// TwinCAT 3 PLC project Printing_Controller
// ProgramVersion: 3.1.4024.0
// libraries:
//   Tc2_Standard, * (Beckhoff Automation GmbH)
//   Tc2_System, * (Beckhoff Automation GmbH)
//   Tc3_Module, * (Beckhoff Automation GmbH)
// project tree:
//   GVLs/ GVL.TcGVL, GVL_IO.TcGVL, GVL_LAP.TcGVL, README.TcGVL
//   / PlcTask.TcTTO
//   POUs/Component/ P_CC1_Enable.TcPOU, P_CP1_Check.TcPOU, P_CP1_Enable.TcPOU
//   POUs/ FB_SetConfigData.TcPOU, FB_GetOutputData.TcPOU, FB_SetOutPutDataToIO.TcPOU, MAIN.TcPOU, P_Control_Mode.TcPOU, P_Laptop_Operate.TcPOU, P_Robot_Operate.TcPOU
//   POUs/Utils/ F_LowpassFilter.TcPOU, F_ScalAnalogOut.TcPOU
// real-time tasks:
//   TASK PlcTask: cycle T#10ms, priority 20, ADS port 350
// I/O:
//   DEVICE Device 1 (EtherCAT), AmsNetId 5.151.68.134.2.1
//     Term 1 (EK1200) [EK1200-5000 EtherCAT Power supply (2A E-Bus)]
//       Term 2 (EL1008) [EL1008 8Ch. Dig. Input 24V, 3ms]
//       Term 3 (EL2008) [EL2008 8Ch. Dig. Output 24V, 0.5A]
//       Term 4 (EL3014) [EL3014 4Ch. Ana. Input 0-20mA DIFF]
//       Term 5 (EL4134) [EL4134 4Ch. Ana. Output -10/+10V, 16bit]
//       Term 6 (EL6631-0010) [EL6631-0010 PROFINET IO Device]
//       Term 7 (EL9011) [EL9011 End Terminal]
// variable links:
//   Printing_Controller/Printing_Controller Instance <-> Device 1 (EtherCAT)/Term 1 (EK1200)/Term 2 (EL1008)
//     PlcTask Inputs/GVL_IO.ibSpare1 <-> Channel 5/Input
//     PlcTask Inputs/GVL_IO.ib_CC1_Button_Mode_Laptop <-> Channel 8/Input
//     PlcTask Inputs/GVL_IO.ib_CC1_Button_Mode_Manual <-> Channel 6/Input
//     PlcTask Inputs/GVL_IO.ib_CC1_Button_Reset <-> Channel 7/Input
//     PlcTask Inputs/GVL_IO.ib_CC1_Safety_Ready <-> Channel 1/Input
//     PlcTask Inputs/GVL_IO.ib_CP1_Drive_Error <-> Channel 4/Input
//     PlcTask Inputs/GVL_IO.ib_CP1_Ready <-> Channel 3/Input
//     PlcTask Inputs/GVL_IO.ib_CP1_Safety_Grid_Mounted <-> Channel 2/Input
//   Printing_Controller/Printing_Controller Instance <-> Device 1 (EtherCAT)/Term 1 (EK1200)/Term 3 (EL2008)
//     PlcTask Outputs/GVL_IO.ob_CC1_Safety_Reset <-> Channel 1/Output
//     PlcTask Outputs/GVL_IO.ob_CP1_Backward <-> Channel 5/Output
//     PlcTask Outputs/GVL_IO.ob_CP1_Forward <-> Channel 4/Output
//     PlcTask Outputs/GVL_IO.ob_CP1_Start <-> Channel 3/Output
//     PlcTask Outputs/GVL_IO.ob_CP1_Stop <-> Channel 2/Output
//   Printing_Controller/Printing_Controller Instance <-> Device 1 (EtherCAT)/Term 1 (EK1200)/Term 4 (EL3014)
//     PlcTask Inputs/GVL_IO.ib_CP1_Actual_Speed <-> AI Standard Channel 1/Value
//   Printing_Controller/Printing_Controller Instance <-> Device 1 (EtherCAT)/Term 1 (EK1200)/Term 5 (EL4134)
//     PlcTask Outputs/GVL_IO.on_CP1_Speed <-> AO Output Channel 1/Analog output

CONFIGURATION Printing_Controller
    RESOURCE PLC ON TwinCAT3
        TASK PlcTask(INTERVAL := T#10ms, PRIORITY := 20);
        PROGRAM MAIN WITH PlcTask : MAIN;
    END_RESOURCE
END_CONFIGURATION

// ---- GVLs/GVL.TcGVL
{attribute 'qualified_only'}
// ***********************************************************************************
//
// USI Mendrisio, Largo Bernasconi 2, CH-6850 Mendrisio
// ETH Zurich, Building HIF E26, Laura-Hezner-Weg 7, CH-8093 Zürich
// 
// ***********************************************************************************
// 
// PROJECT     :  Clay Printing Controller
// FUNCTION    :  Global varable
// AUTHOR      :  WeiTing Chen
// EMAIL       :  chen@mesh.ch
// Copyright   :  USI FMAA Mendrisio(CH) 2025
//
// ***********************************************************************************


VAR_GLOBAL
	
	// Controller 1
	b_mode_manual : BOOL;
	b_mode_laptop : BOOL; 
	b_mode_robot : BOOL;  
	
	b_CC1_enable :BOOL;
	b_CC1_power_on: BOOL;
	s_current_mode: STRING;
	
	// Machine 1
	// Machine 2
	
	// Concrete Pump 1
	b_CP1_Check_On : BOOL;
	b_CP1_is_run : BOOL;
	b_CP1_is_ready : BOOL;	
	b_CP1_power_on :BOOL;
	b_CP1_safety_grid_on : BOOL;
	b_CP1_drive_error :BOOL;
	
	
	// Config
	// Concrete Pump 1
	f_CP1_Max_Flowrate : REAL;
	f_CP1_Check_Flowrate : REAL;
	t_CP1_Check_Duration : TIME;
 	n_CP1_Flush_Flowrate :REAL;	
	
END_VAR

// ---- GVLs/GVL_IO.TcGVL
{attribute 'qualified_only'}

// ***********************************************************************************
//
// USI Mendrisio, Largo Bernasconi 2, CH-6850 Mendrisio
// ETH Zurich, Building HIF E26, Laura-Hezner-Weg 7, CH-8093 Zürich
//
// ***********************************************************************************
//
// PROJECT     :  Clay Printing Controller
// FUNCTION    :  Global Hareware IO
// AUTHOR      :  WeiTing Chen
// EMAIL       :  chen@mesh.ch
// Copyright   :  USI FMAA Mendrisio(CH) 2025
//
// ***********************************************************************************

VAR_GLOBAL

	// ***** HARDWARE INPUT ******

	// Concrete Controller 1
	// This once install the safety gate, we can start to do read from it.
	ib_CC1_Safety_Ready_NOT_IMP AT %I*: BOOL;  // DI1
	ib_CC1_Safety_Ready:BOOL;
	ib_CC1_Button_Mode_Manual   AT %I*: BOOL;  // DI6
	ib_CC1_Button_Mode_Laptop   AT %I*: BOOL;  // DI8
	ib_CC1_Button_Reset         AT %I*: BOOL;  // DI7

	// Concrete Pump 1
	ib_CP1_Safety_Grid_Mounted  AT %I*: BOOL;  // DI2
	ib_CP1_Ready                AT %I*: BOOL;  // DI3
	ib_CP1_Drive_Error          AT %I*: BOOL;  // DI4
	ib_CP1_Actual_Speed         AT %I*: INT;   // AI1

	// Spare Slot
	ibSpare1 AT %I*: BOOL;  //DI5
	inSpare2 AT %I*: INT;   //AI2
	inSpare3 AT %I*: INT;   //AI3
	inSpare4 AT %I*: INT;   //AI4


	// ***** HARDWARE OUTPUT ******

	// Concrete Controller 1
	ob_CC1_Safety_Reset AT %Q*: BOOL;  //DO1

	// Concrete Pump 1
	ob_CP1_Start    AT %Q*: BOOL;  //DO3
	ob_CP1_Stop     AT %Q*: BOOL;  //DO2
	ob_CP1_Forward  AT %Q*: BOOL;  //DO4
	ob_CP1_Backward AT %Q*: BOOL;  //DO5
	on_CP1_Speed    AT %Q*: INT;   //AO1
	// just for testing, if not working after we can delete it.
	on_CP1_Speed_test    AT %Q*: INT;   //AOTemp

	// Spare Slot
	obSpare6 AT %Q*: BOOL;  //DO6
	obSpare7 AT %Q*: BOOL;  //DO7
	obSpare8 AT %Q*: BOOL;  //DO8

	onSpare2 AT %Q*: INT;   //AO2
	onSpare3 AT %Q*: INT;   //AO3
	onSpare4 AT %Q*: INT;   //AO4

END_VAR

// ---- GVLs/GVL_LAP.TcGVL
{attribute 'qualified_only'}

// ***********************************************************************************
//
// USI Mendrisio, Largo Bernasconi 2, CH-6850 Mendrisio
// ETH Zurich, Building HIF E26, Laura-Hezner-Weg 7, CH-8093 Zürich
//
// ***********************************************************************************
//
// PROJECT     :  Clay Printing Controller
// FUNCTION    :  Global Laptop IO wrapper
// AUTHOR      :  WeiTing Chen
// EMAIL       :  chen@mesh.ch
// Copyright   :  USI FMAA Mendrisio(CH) 2025
//
// ***********************************************************************************

VAR_GLOBAL
	
	CONCRETE_CONTROLLER: STRING := 'Controller'; //*****
	b_Operate_mode_manual             : BOOL;
	b_Operate_mode_laptop             : BOOL;
	b_Operate_mode_robot              : BOOL;
	b_Concrete_Controller_enable      : BOOL;
	b_Concrete_Controller_reset       : BOOL;
	b_Concrete_Controller_power_on    : BOOL;
	n_Concrete_Controller_current_mode: INT;
	
	CONCRETE_PUMP: STRING := 'CONCRETE_PUMP'; //*****
	// Concrete Pump
	// input
	
	b_Concrete_Pump_Power_On   : BOOL;  // Power On
	b_Concrete_Pump_Forward_On : BOOL;  // Forward ON
	b_Concrete_Pump_Backward_On: BOOL;  // Backward ON
	
	b_Concrete_Pump_Flush_On      : BOOL;  // FLUSH MODE ON
	n_Concrete_Pump_Flush_Flowrate: REAL;  // READ [l/min]
	
	b_Concrete_Pump_Check_On      : BOOL;       // CHECK MODE ON
	
	// TODO: Need to check the range of flowrate
	f_Concrete_Pump_Check_Flowrate: REAL;       // [O tp 24 l/min]
	n_Concrete_Pump_Check_Duration: INT := 15;  // [s]
	
	f_Concrete_Pump_Set_Flowrate : REAL;          // [0 to 24 l/min]
	f_Concrete_Pump_dosing_volume: REAL := 0.32;  // calibrated XXXXX
	n_Concrete_Pump_Max_Speed    : INT := 75;     // calibrated XXXXX
	n_Concrete_Pump_Set_Speed    : INT;           // WRITE VALUE From 0 to 75 [rpm]
	
	
	b_CP1_is_run        : BOOL;
	b_CP1_is_ready      : BOOL;
	b_CP1_power_on      : BOOL;
	b_CP1_safety_grid_on: BOOL;
	b_CP1_drive_error   : BOOL;
	
	
	f_CP1_status_torque :REAL;
	f_CP1_status_speed: REAL;
	
	// Other
	Admixture_Pump_1: STRING := 'Admixture Pump (AP1)'; //*****

END_VAR

// ---- GVLs/README.TcGVL
{attribute 'qualified_only'}
// ***********************************************************************************
//
// USI Mendrisio, Largo Bernasconi 2, CH-6850 Mendrisio
// ETH Zurich, Building HIF E26, Laura-Hezner-Weg 7, CH-8093 Zürich
//
// ***********************************************************************************
//
// PROJECT     :  Clay Printing Controller
// FUNCTION    :  README
// AUTHOR      :  WeiTing Chen
// EMAIL       :  chen@mesh.ch
// Copyright   :  USI FMAA Mendrisio(CH) 2025
//
// ***********************************************************************************

VAR_GLOBAL
(*
Set the IP with XXXXXXXX

File description
GVL(GVL : Global variables)
GVL_IO(GVL_IO : IO)
GVL_LAP(GVL_LAP : variables for control via laptop)

Data Type Prefix
ib = Input Bool   / ob = Output Bool
if = Input float  / of = Output float (REAL, LREAL)
in = Input numeric/ on = Output numeric
(INT, SINT, USINT, UNIT, DINT, UDINT, BYTE, WORD, DWORD, LWORD, XINT, UXINT, XWORD)
t = Time (TON)
s = String

Naming Shortcuts
CC1 = Concrete Controller
CP1 = Concrete Pump
PN = Profinet with Roboter

*)
END_VAR

// ---- POUs/MAIN.TcPOU
PROGRAM MAIN
VAR
END_VAR


// ***********************************************************************************
//
// USI Mendrisio, Largo Bernasconi 2, CH-6850 Mendrisio
// ETH Zurich, Building HIF E26, Laura-Hezner-Weg 7, CH-8093 Zürich
//
// ***********************************************************************************
//
// PROJECT     :  Clay Printing Controller
// FUNCTION    :  Main
// AUTHOR      :  WeiTing Chen
// EMAIL       :  chen@mesh.ch
// Copyright   :  USI FMAA Mendrisio(CH) 2025
//
// ***********************************************************************************


// Control Mode select
P_Control_Mode();

// Operation Mode select
// TODO: Implementation of the operation mode. Now everything services as laptop mode.
IF GVL.b_mode_laptop THEN
	P_Laptop_Operate();
ELSIF GVL.b_mode_robot THEN
	P_Laptop_Operate();
ELSIF GVL.b_mode_manual THEN
	P_Laptop_Operate();
END_IF

END_PROGRAM

// ---- POUs/P_Control_Mode.TcPOU
PROGRAM P_Control_Mode
VAR
END_VAR


// ***********************************************************************************
//
// USI Mendrisio, Largo Bernasconi 2, CH-6850 Mendrisio
// ETH Zurich, Building HIF E26, Laura-Hezner-Weg 7, CH-8093 Zürich
//
// ***********************************************************************************
//
// PROJECT     :  Clay Printing Controller
// FUNCTION    :  Control mode selection
// AUTHOR      :  WeiTing Chen
// EMAIL       :  chen@mesh.ch
// Copyright   :  USI FMAA Mendrisio(CH) 2025
//
// ***********************************************************************************


GVL.b_mode_manual := GVL_IO.ib_CC1_Button_Mode_Manual;
GVL.b_mode_laptop := GVL_IO.ib_CC1_Button_Mode_Laptop;
GVL.b_mode_robot := False;

IF GVL.b_mode_manual THEN
	GVL.s_current_mode := 'Controller';
ELSIF GVL.b_mode_laptop  THEN
	GVL.s_current_mode := 'Laptop';
ELSIF NOT GVL.b_mode_manual AND NOT GVL.b_mode_laptop THEN
	GVL.s_current_mode := 'Robot';
	GVL.b_mode_robot := TRUE;
ELSE
	GVL.s_current_mode := 'None';

END_IF

END_PROGRAM

// ---- POUs/P_Laptop_Operate.TcPOU
PROGRAM P_Laptop_Operate
VAR
	SafetyReset 	: bool;
	b_Enable		: BOOL;
	b_Reset			: BOOL;

	fb_SetOutputDataToIO : FB_SetOutputDataToIO;
	fb_getOutputData : FB_GetOutputData;
	fb_setConfig : FB_SetConfigData;

	b_Safety_Reset : BOOL;
	b_Timer_Rest : BOOL;
	t_CC1_Time_Safety_Rest : TIME :=T#5S; //wait 5s for controller restart
	fb_CC1_Trigger_Safety_On : R_TRIG;
	fb_CC1_Trigger_Safety_Off : R_TRIG;
	fb_CC1_Timer_Safety: TON;

END_VAR


// ***********************************************************************************
//
// USI Mendrisio, Largo Bernasconi 2, CH-6850 Mendrisio
// ETH Zurich, Building HIF E26, Laura-Hezner-Weg 7, CH-8093 Zürich
//
// ***********************************************************************************
//
// PROJECT     :  Clay Printing Controller
// FUNCTION    :  Control mode selection
// AUTHOR      :  WeiTing Chen
// EMAIL       :  chen@mesh.ch
// Copyright   :  USI FMAA Mendrisio(CH) 2025
//
// ***********************************************************************************

// Controller reset trigger
b_Timer_Rest:=GVL_LAP.b_Concrete_Controller_reset;

fb_CC1_Timer_Safety(
					IN:=b_Timer_Rest,
					PT:=t_CC1_Time_Safety_Rest);

fb_CC1_Trigger_Safety_On(clk:=fb_CC1_Timer_Safety.IN);
fb_CC1_Trigger_Safety_Off(clk:=fb_CC1_Timer_Safety.Q);
//b_Safety_Reset:=FALSE;
IF fb_CC1_Trigger_Safety_On.Q THEN
	b_Safety_Reset:=TRUE;
END_IF
IF fb_CC1_Trigger_Safety_Off.Q THEN
	b_Safety_Reset:=FALSE;
	GVL_LAP.b_Concrete_Controller_reset:=FALSE;
END_IF
GVL_IO.ob_CC1_Safety_Reset:= b_Safety_Reset OR GVL_IO.ib_CC1_Button_Reset;

// Concrete Controller enable
P_CC1_Enable( b_set_run:= GVL_LAP.b_Concrete_Controller_enable );


//***********************************************************************************
// Set Process Configuration
//***********************************************************************************

fb_setConfig(
// Geneal
// Concrete Controller

// Concrete Pump
_f_CP1_Max_Flowrate   := INT_TO_REAL(GVL_LAP.n_Concrete_Pump_Max_Speed) * GVL_LAP.f_Concrete_Pump_dosing_volume,
_f_CP1_Check_Flowrate := GVL_LAP.f_Concrete_Pump_Check_Flowrate,
_t_CP1_Check_Duration := INT_TO_TIME(GVL_LAP.n_Concrete_Pump_Check_Duration)*1000,

);

//***********************************************************************************
// Setup IO data to PLC
//***********************************************************************************
fb_SetOutputDataToIO(

	// Concrete Pump
	b_CP1_Forward_On       := GVL_LAP.b_Concrete_Pump_Forward_On,
	b_CP1_Backward_On      := GVL_LAP.b_Concrete_Pump_Backward_On,
	b_CP1_Flush_On         := GVL_LAP.b_Concrete_Pump_Flush_On,
	b_CP1_Check_On         := GVL_LAP.b_Concrete_Pump_Check_On,
	n_CP_Flowrate_mode     := TRUE,
	n_CP1_Operate_Flowrate := REAL_TO_UDINT(GVL_LAP.f_Concrete_Pump_Set_Flowrate*100),
	n_CP1_Check_Flowrate   := REAL_TO_UDINT(GVL_LAP.f_Concrete_Pump_Check_Flowrate*100),
	n_CP1_Flush_Flowrate   := REAL_TO_UDINT(GVL_LAP.n_Concrete_Pump_Flush_Flowrate*100),
	f_dosing_volume        := REAL_TO_INT(GVL_LAP.f_concrete_pump_dosing_volume*100),
	n_cp1_max_speed        := GVL_LAP.n_concrete_pump_max_speed,
	n_cp1_target_speed     := GVL_LAP.n_concrete_pump_set_speed,

  //
	);


//***********************************************************************************
// Concrete Pump
//***********************************************************************************

// concrete pump power control is from pump itself
P_CP1_Enable();
P_CP1_Check(b_set_run := fb_SetOutputDataToIO.b_CP1_Forward_On,
			b_check_mode_on  := fb_SetOutputDataToIO.b_CP1_Check_On,
			t_check_duration := fb_setConfig._t_CP1_Check_Duration,
			);


//***********************************************************************************
// Other Pump
//***********************************************************************************

// Put Other pump control here


//***********************************************************************************
// Get out put data from PLC
//***********************************************************************************
fb_getOutputData(

	//CC1
	b_mode_manual := GVL_LAP.b_Operate_mode_manual,
	b_mode_laptop := GVL_LAP.b_Operate_mode_laptop,
	b_mode_robot   := GVL_LAP.b_Operate_mode_robot,
	b_CC1_power_on := GVL_LAP.b_Concrete_Controller_power_on,
	n_current_mode := GVL_LAP.n_Concrete_Controller_current_mode,

	//CP1
	b_CP1_is_run   := GVL_LAP.b_CP1_is_run,
	b_CP1_is_ready := GVL_LAP.b_CP1_is_ready,

	b_CP1_power_on       := GVL_LAP.b_CP1_power_on,
	b_CP1_safety_grid_on := GVL_LAP.b_CP1_safety_grid_on,
	b_CP1_drive_error    := GVL_LAP.b_CP1_drive_error,
	
	f_CP1_status_torque := GVL_LAP.f_CP1_status_torque,
	f_CP1_status_speed := GVL_LAP.f_CP1_status_speed,

);

END_PROGRAM

// ---- POUs/FB_SetOutPutDataToIO.TcPOU
FUNCTION_BLOCK  FB_SetOutPutDataToIO
VAR_INPUT

	// Concrete Pump
	b_CP1_Forward_On : BOOL;
	b_CP1_Backward_On : BOOL;
	b_CP1_Flush_On :BOOL;
	b_CP1_Check_On : BOOL;
	n_CP_Flowrate_mode : BOOL;
	n_CP1_Operate_Flowrate : UDINT;
	n_CP1_Check_Flowrate : UDINT;
	n_CP1_Flush_Flowrate : UDINT;
	f_dosing_volume:INT;

	n_CP1_max_speed : INT ;  // rpm
	n_CP1_target_speed: INT; // rpm

	// Example for AP1
	(*
	b_AP1_Power_On : BOOL;
	b_AP1_Run : BOOL;
	b_AP1_Flush_On :BOOL;
	b_AP1_Check_On :BOOL;

	n_AP1_Flowrate_mode : BOOL;
	n_AP1_Max_Flowrate : INT;
	n_AP1_Operate_Flowrate : UDINT;
	n_AP1_Check_Flowrate : UDINT;
	n_AP1_Flush_Flowrate : UDINT;
	n_AP1_Dosing_factor : INT;
	*)


END_VAR
VAR_OUTPUT
END_VAR
VAR
	// Condition
	_n_temp_flowrate_CP1 : UDINT;
	_n_temp_speed_CP1: INT;

END_VAR

// ***********************************************************************************
//
// USI Mendrisio, Largo Bernasconi 2, CH-6850 Mendrisio
// ETH Zurich, Building HIF E26, Laura-Hezner-Weg 7, CH-8093 Zürich
//
// ***********************************************************************************
//
// PROJECT     :  Clay Printing Controller
// FUNCTION    :  Set data to IO and process (Custom function block)
// AUTHOR      :  WeiTing Chen
// EMAIL       :  chen@mesh.ch
// Copyright   :  USI FMAA Mendrisio(CH) 2025
//
// ***********************************************************************************


// ***********************************************************************************
// Concrete Pump 1
// ***********************************************************************************


// Start
IF  P_CP1_Enable.n_Step=20 THEN
	GVL_IO.ob_CP1_Start:=TRUE;
ELSE
	GVL_IO.ob_CP1_Start:=FALSE;
END_IF

// Stop
IF  P_CP1_Enable.n_Step=40 THEN
	GVL_IO.ob_CP1_Stop:=TRUE;
ELSE
	GVL_IO.ob_CP1_Stop:=FALSE;
END_IF

GVL_IO.ob_CP1_Forward := b_CP1_Forward_On; // Forward
GVL_IO.ob_CP1_Backward := b_CP1_Backward_On; // Backward

// Set speed for pump
IF b_CP1_Flush_On THEN
	//
	// Process speed for flushing or filling the pipe
	 _n_temp_flowrate_CP1:=n_CP1_Flush_Flowrate;
ELSIF P_CP1_Check.n_Step=20 OR P_CP1_Check.n_Step=25 THEN
	//
	// Check Flowrate for pump
	_n_temp_flowrate_CP1 :=n_CP1_Check_Flowrate;
ELSE
	//
	// Process speed for pump
	_n_temp_flowrate_CP1 :=n_CP1_Operate_Flowrate;
END_IF


// Concrete pump speed  0 (0V) to 75 rpm (10V)
IF NOT n_CP_Flowrate_mode THEN
	// set from rpm
	GVL_IO.on_CP1_Speed:=F_ScalAnalogOut(
		n_Input:= INT_TO_UDINT(n_CP1_target_speed),
		n_InMin:= 0,
		n_InMax:= INT_TO_UDINT(n_CP1_max_speed),
		n_OutMin:= 0,
		n_OutMax:= 32767);
ELSE
	// set from flowrate
	GVL_IO.on_CP1_Speed:=F_ScalAnalogOut(
		n_Input:= _n_temp_flowrate_CP1,
		n_InMin:= 0,
		n_InMax:= INT_TO_UDINT(n_CP1_max_speed*f_dosing_volume),
		n_OutMin:= 0,
		n_OutMax:= 32767);
END_IF


//***********************************************************************************
// Other Pump
//***********************************************************************************

END_FUNCTION_BLOCK

// ---- POUs/Component/P_CP1_Enable.TcPOU
PROGRAM P_CP1_Enable
VAR_INPUT
	// INT 
	n_Step: INT := 0;	
END_VAR
VAR
	// BOOL 
	b_Condition: BOOL;
	b_No_Emergency_Stop:BOOL :=TRUE;

	//
	// Timer 
	t_CP1_Puls_Enable: TON;	
	t_CP1_Puls_Disable: TON;	
	
END_VAR

// ***********************************************************************************
//
// USI Mendrisio, Largo Bernasconi 2, CH-6850 Mendrisio
// ETH Zurich, Building HIF E26, Laura-Hezner-Weg 7, CH-8093 Zürich
//
// ***********************************************************************************
//
// PROJECT     :  Clay Printing Controller
// FUNCTION    :  Step chain for concrete pump enable
// AUTHOR      :  WeiTing Chen
// EMAIL       :  chen@mesh.ch
// Copyright   :  USI FMAA Mendrisio(CH) 2025
//
// ***********************************************************************************

// Ignore emergency stop
b_No_Emergency_Stop:=TRUE;

//
// Initalization
IF n_Step=0 THEN
	//
	// Check condition 
	b_Condition:=TRUE;
	//
	// Do step
	IF b_Condition THEN
		b_Condition:=FALSE;
		n_Step:=10;
	END_IF
END_IF

//
// Check grid mounted and no errors 
IF n_Step=10 THEN
	//
	// Check condition 
	b_Condition:= GVL_IO.ib_CP1_Safety_Grid_Mounted AND NOT GVL_IO.ib_CP1_Drive_Error;
	//
	// Do step
	IF b_Condition AND b_No_Emergency_Stop THEN
		b_Condition:=FALSE;
		n_Step:=20;
	END_IF
END_IF

//
// Send enable to pump
IF n_Step=20 THEN
	//
	// Check condition 
	b_Condition:=t_CP1_Puls_Enable.Q;
	//
	// Do step
	IF b_Condition AND b_No_Emergency_Stop THEN
		b_Condition:=FALSE;
		n_Step:=30;
	END_IF
END_IF

//
// Pump enabled checking for errors or grid removed
IF n_Step=30 THEN
	//
	// Check condition 
	b_Condition:= NOT GVL_IO.ib_CP1_Safety_Grid_Mounted OR GVL_IO.ib_CP1_Drive_Error;
	//
	// Do step
	IF b_Condition THEN
		b_Condition:=FALSE;
		n_Step:=40;
	END_IF
END_IF

//
// Send disable to pump
IF n_Step=40 THEN
	//
	// Check condition 
	b_Condition:=t_CP1_Puls_Disable.Q;
	//
	// Do step
	IF b_Condition AND b_No_Emergency_Stop THEN
		b_Condition:=FALSE;
		n_Step:=50;
	END_IF
END_IF

//
// Return to step 10 
IF n_Step=50 THEN
	//
	// Check condition 
	b_Condition:=TRUE;
	//
	// Do step
	IF b_Condition THEN
		b_Condition:=FALSE;
		n_Step:=10;
	END_IF
END_IF

// ****************************************
// Timer
// ****************************************
t_CP1_Puls_Enable(
	IN:=n_Step=20,
	PT:=T#200MS);

t_CP1_Puls_Disable(
	IN:=n_Step=40,
	PT:=T#200MS);

END_PROGRAM

// ---- POUs/Component/P_CP1_Check.TcPOU
PROGRAM P_CP1_Check
VAR
END_VAR

END_PROGRAM

// ---- POUs/Utils/F_ScalAnalogOut.TcPOU
FUNCTION F_ScalAnalogOut :INT
VAR_INPUT
	n_Input:UDINT;
	n_InMin:UDINT;
	n_InMax:UDINT;
	n_OutMin:UDINT;
	n_OutMax:UDINT;

END_VAR
VAR
	f_Input:REAL;
	f_InMin:REAL;
	f_InMax:REAL;
	f_OutMin:REAL;
	f_OutMax:REAL;
	f_DeltaIn:REAL;
	f_DeltaOut:REAL;
END_VAR

// ***********************************************************************************
//
// USI Mendrisio, Largo Bernasconi 2, CH-6850 Mendrisio
// ETH Zurich, Building HIF E26, Laura-Hezner-Weg 7, CH-8093 Zürich
//
// ***********************************************************************************
//
// PROJECT     :  Clay Printing Controller
// FUNCTION    :  Func scale analogue output
// AUTHOR      :  WeiTing Chen
// EMAIL       :  chen@mesh.ch
// Copyright   :  USI FMAA Mendrisio(CH) 2025
//
// ***********************************************************************************
//
// Check plausibility 

IF f_Input > f_InMax THEN
	f_Input := f_InMax;
END_IF

IF f_InMax = f_InMin THEN	
	//
	// Not plausible output fix value
	F_ScalAnalogOut := 0;
ELSE
	// Check the input data is lager than maximum
	IF f_Input > f_InMax THEN
		f_Input := f_InMax;
	END_IF
	//
	// Plausible calculate output 
	f_DeltaIn:=f_InMax-f_InMin;
	f_DeltaOut:=f_OutMax-f_OutMin;
	F_ScalAnalogOut :=REAL_TO_INT((f_DeltaOut/f_DeltaIn)*(f_Input-f_InMin));	
END_IF

END_FUNCTION

// ---- POUs/FB_GetOutputData.TcPOU
FUNCTION_BLOCK  FB_GetOutputData
VAR_INPUT
	//Gerenal
	b_Output_number_REALMode : BOOL;
END_VAR

VAR_IN_OUT
	//CC1
	b_mode_manual : BOOL;
	b_mode_laptop : BOOL;
	b_mode_robot : BOOL;
	b_CC1_power_on : BOOL;
	n_current_mode : INT;

	//CP1
	b_CP1_is_run : BOOL;
	b_CP1_is_ready : BOOL;
	b_CP1_power_on :BOOL;
	b_CP1_safety_grid_on : BOOL;
	b_CP1_drive_error :BOOL;

	f_CP1_status_torque : REAL;
	f_CP1_status_speed : REAL;
	
END_VAR
VAR_OUTPUT
END_VAR
VAR
END_VAR

// ***********************************************************************************
//
// USI Mendrisio, Largo Bernasconi 2, CH-6850 Mendrisio
// ETH Zurich, Building HIF E26, Laura-Hezner-Weg 7, CH-8093 Zürich
//
// ***********************************************************************************
//
// PROJECT     :  Clay Printing Controller
// FUNCTION    :  Get data From IO and process (Custom function block)
// AUTHOR      :  WeiTing Chen
// EMAIL       :  chen@mesh.ch
// Copyright   :  USI FMAA Mendrisio(CH) 2025
//
// ***********************************************************************************


// General
b_mode_manual := GVL.b_mode_manual;
b_mode_laptop := GVL.b_mode_laptop;
b_mode_robot := GVL.b_mode_robot;
b_CC1_power_on := GVL.b_CC1_power_on;

IF GVL.s_current_mode = 'Controller'THEN
	n_current_mode := 1;
ELSIF GVL.s_current_mode = 'Laptop' THEN
	n_current_mode := 2;
ELSIF GVL.s_current_mode = 'Robot' THEN
	n_current_mode := 3;
ELSE
	n_current_mode := 4;
END_IF


// Concrete Pump
// Status
GVL.b_CP1_Is_Run := GVL_IO.ob_CP1_Forward;
b_CP1_is_run := GVL.b_CP1_Is_Run;

GVL.b_CP1_is_ready := GVL_IO.ib_CP1_Ready;
b_CP1_is_ready := GVL.b_CP1_is_ready;

GVL.b_CP1_power_on :=  GVL_IO.ib_CP1_Ready;
b_CP1_power_on := GVL.b_CP1_power_on;

GVL.b_CP1_safety_grid_on := GVL_IO.ib_CP1_Safety_Grid_Mounted;
b_CP1_safety_grid_on := GVL.b_CP1_safety_grid_on;

GVL.b_CP1_drive_error := GVL_IO.ib_CP1_Drive_Error;
b_CP1_drive_error := GVL.b_CP1_drive_error;


// Torque
// TODO: make it from actual speed value.

IF b_Output_number_REALMode THEN
	f_CP1_status_torque := F_LowpassFilter(GVL_IO.ib_CP1_Actual_Speed)*0.1;
	f_CP1_status_speed := F_LowpassFilter(GVL_IO.ib_CP1_Actual_Speed)*0.1;

ELSE
	f_CP1_status_speed := F_LowpassFilter(GVL_IO.ib_CP1_Actual_Speed);
	f_CP1_status_speed := F_LowpassFilter(GVL_IO.ib_CP1_Actual_Speed);
END_IF

// Temperature
// pass
// Pressure
// pass

END_FUNCTION_BLOCK

// ---- POUs/Utils/F_LowpassFilter.TcPOU
FUNCTION F_LowpassFilter : REAL
VAR_INPUT
	rValueIn	:REAL;
END_VAR
VAR
	rValue_In	:REAL;
	rValue_New	:REAL;	
	rValue_Old	:REAL;
	rFactor	    :REAL := 0.1; // 10% old new value			

END_VAR

// ***********************************************************************************
//
// USI Mendrisio, Largo Bernasconi 2, CH-6850 Mendrisio
// ETH Zurich, Building HIF E26, Laura-Hezner-Weg 7, CH-8093 Zürich
//
// ***********************************************************************************
//
// PROJECT     :  Clay Printing Controller
// FUNCTION    :  F_LowpassFilter
// AUTHOR      :  WeiTing Chen
// EMAIL       :  chen@mesh.ch
// Copyright   :  USI FMAA Mendrisio(CH) 2025
//
// ***********************************************************************************

rValue_In := rValueIn;

IF rValue_Old = 0 THEN;
	rValue_Old := rValue_In;
	rValue_New := ((1-rFactor)*rValue_Old) + (rFactor*rValue_In);
ELSE
	rValue_Old := rValue_New;
	rValue_New := ((1-rFactor)*rValue_Old) + (rFactor*rValue_In);
END_IF


// Read IO in and out
F_LowpassFilter := rValue_New;

END_FUNCTION

// ---- POUs/FB_SetConfigData.TcPOU
FUNCTION_BLOCK FB_SetConfigData
VAR_INPUT
	// Gerenal
	// Concrete Controller

	// Concrete Pump
	_f_CP1_Max_Flowrate : REAL;
	_f_CP1_Check_Flowrate : REAL;
	_t_CP1_Check_Duration : TIME;

END_VAR
VAR_OUTPUT
END_VAR
VAR
END_VAR

// ***********************************************************************************
//
// USI Mendrisio, Largo Bernasconi 2, CH-6850 Mendrisio
// ETH Zurich, Building HIF E26, Laura-Hezner-Weg 7, CH-8093 Zürich
//
// ***********************************************************************************
//
// PROJECT     :  Clay Printing Controller
// FUNCTION    :  Set all default/constant data for the process (Custom function block)
// AUTHOR      :  WeiTing Chen
// EMAIL       :  chen@mesh.ch
// Copyright   :  USI FMAA Mendrisio(CH) 2025
//
// ***********************************************************************************

// Setter for the components Config
// Concrete Controller (CC1)

// Concrete Pump 1
GVL.f_CP1_Max_Flowrate := _f_CP1_Max_Flowrate;
GVL.f_CP1_Check_Flowrate := _f_CP1_Check_Flowrate;
GVL.t_CP1_Check_Duration := _t_CP1_Check_Duration;
GVL.n_CP1_Flush_Flowrate := (_f_CP1_Max_Flowrate) / 2;

END_FUNCTION_BLOCK

// ---- POUs/Component/P_CC1_Enable.TcPOU
PROGRAM P_CC1_Enable
VAR_INPUT
	n_Step: INT := 0;	
	b_set_run : BOOL;
END_VAR
VAR
	//
	// BOOL 
	b_Condition: BOOL;
	b_No_Emergency_Stop:BOOL :=TRUE;
	
END_VAR

// ***********************************************************************************
//
// USI Mendrisio, Largo Bernasconi 2, CH-6850 Mendrisio
// ETH Zurich, Building HIF E26, Laura-Hezner-Weg 7, CH-8093 Zürich
//
// ***********************************************************************************
//
// PROJECT     :  Clay Printing Controller
// FUNCTION    :  Step chain for controller enable
// AUTHOR      :  WeiTing Chen
// EMAIL       :  chen@mesh.ch
// Copyright   :  USI FMAA Mendrisio(CH) 2025
//
// ***********************************************************************************

//
// Ignore emergency stop
b_No_Emergency_Stop:=TRUE;

//
// Initalization
IF n_Step=0 THEN
	//
	// Check condition 
	b_Condition:=TRUE;
	//
	// Do step
	IF b_Condition THEN
		b_Condition:=FALSE;
		n_Step:=10;
	END_IF
END_IF

//
// Wait for start
IF n_Step=10 THEN
	//
	// Check condition 
	b_Condition:= GVL_IO.ib_CC1_Safety_Ready AND b_set_run;
	//
	// Do step
	IF b_Condition AND b_No_Emergency_Stop THEN
		b_Condition:=FALSE;
		n_Step:=20;
	END_IF
END_IF

//
// Reserve
IF n_Step=20 THEN
	//
	// Check condition 
	b_Condition:=TRUE;
	//
	// Do step
	IF b_Condition AND b_No_Emergency_Stop THEN
		b_Condition:=FALSE;
		n_Step:=30;
	END_IF
END_IF

//
// Run 
IF n_Step=30 THEN
	//
	// Check condition 
	b_Condition:= NOT GVL_IO.ib_CC1_Safety_Ready OR NOT b_set_run;
	//
	// Do step
	IF b_Condition THEN
		b_Condition:=FALSE;
		n_Step:=40;
	END_IF
END_IF

//
//
IF n_Step=40 THEN
	//
	// Check condition 
	b_Condition:=TRUE;
	//
	// Do step
	IF b_Condition AND b_No_Emergency_Stop THEN
		b_Condition:=FALSE;
		n_Step:=50;
	END_IF
END_IF

//
// Return to step 10 
IF n_Step=50 THEN
	//
	// Check condition 
	b_Condition:=TRUE;
	//
	// Do step
	IF b_Condition THEN
		
		b_Condition:=FALSE;
		n_Step:=10;
	END_IF
END_IF

//
// Mixer run
GVL.b_CC1_power_on:=n_Step=30;

END_PROGRAM

// ---- POUs/P_Robot_Operate.TcPOU
PROGRAM P_Robot_Operate
VAR
END_VAR

//No implements

END_PROGRAM
